// LS Electric XG5000 project: 과년66_1_3
// PLC NewPLC
// module base 0 slot 0: 입출력 모듈:XBC-DR20S (DC 24V 입력 12점, 릴레이 출력 8점)

PROGRAM NewProgram (task: 스캔 프로그램)

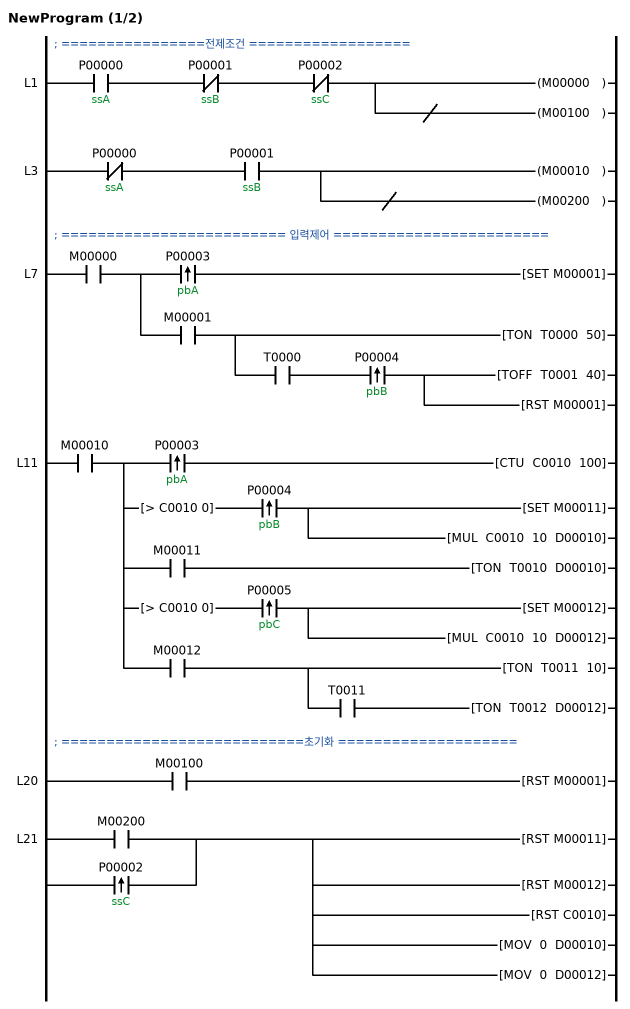
// ================전제조건 ==================
; L1
LOAD      P00000	// ssA
AND NOT   P00001	// ssB
AND NOT   P00002	// ssC
OUT       M00000
NOT
OUT       M00100
; L3
LOAD NOT  P00000	// ssA
AND       P00001	// ssB
OUT       M00010
NOT
OUT       M00200
// ========================= 입력제어 ========================
; L7
LOAD      M00000
MPUSH
ANDP      P00003	// pbA
SET       M00001
MPOP
AND       M00001
TON       T0000 50
AND       T0000
ANDP      P00004	// pbB
TOFF      T0001 40
RST       M00001
; L11
LOAD      M00010
MPUSH
ANDP      P00003	// pbA
CTU       C0010 100
MLOAD
AND>      C0010 0
ANDP      P00004	// pbB
SET       M00011
MUL       C0010 10 D00010
MLOAD
AND       M00011
TON       T0010 D00010
MLOAD
AND>      C0010 0
ANDP      P00005	// pbC
SET       M00012
MUL       C0010 10 D00012
MPOP
AND       M00012
TON       T0011 10
AND       T0011
TON       T0012 D00012
// ===========================초기화 ====================
; L20
LOAD      M00100
RST       M00001
; L21
LOAD      M00200
ORP       P00002	// ssC
RST       M00011
RST       M00012
RST       C0010
MOV       0 D00010
MOV       0 D00012

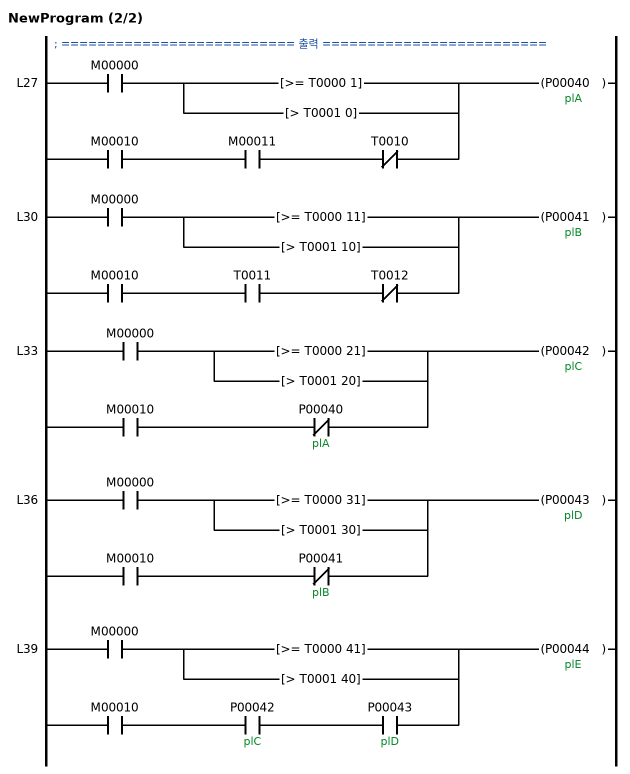
// ========================== 출력 =========================
; L27
LOAD      M00000
LOAD>=    T0000 1
OR>       T0001 0
AND LOAD
LOAD      M00010
AND       M00011
AND NOT   T0010
OR LOAD
OUT       P00040	// plA
; L30
LOAD      M00000
LOAD>=    T0000 11
OR>       T0001 10
AND LOAD
LOAD      M00010
AND       T0011
AND NOT   T0012
OR LOAD
OUT       P00041	// plB
; L33
LOAD      M00000
LOAD>=    T0000 21
OR>       T0001 20
AND LOAD
LOAD      M00010
AND NOT   P00040	// plA
OR LOAD
OUT       P00042	// plC
; L36
LOAD      M00000
LOAD>=    T0000 31
OR>       T0001 30
AND LOAD
LOAD      M00010
AND NOT   P00041	// plB
OR LOAD
OUT       P00043	// plD
; L39
LOAD      M00000
LOAD>=    T0000 41
OR>       T0001 40
AND LOAD
LOAD      M00010
AND       P00042	// plC
AND       P00043	// plD
OR LOAD
OUT       P00044	// plE